ABB RobotStudio station: Minor Project_Kundan_Singh_48849855.rspag

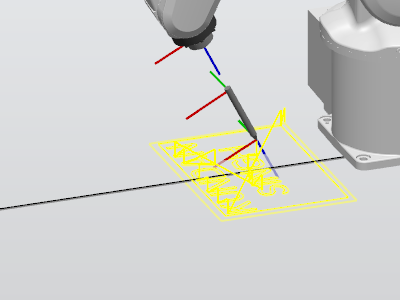
--- station ---
Station Minor Project Kundan1_4 (saved by RobotStudio 23.2.10395.0)
Controller Controller8, task T_ROB1: task frame (RAPID world) sits at (0, -187, 16) mm in the station
Controller Controller8
  mechanical unit ROB_1: IRB120_3_58__01, 6 joints, base frame (0, 0, 0) mm
Layout (positions relative to the parent item):
  - IRB120_3_58__01 [mechanism, from %ABB.RobotStudio.Models.IRB120%\IRB120_3_58_G_01.rslib] at (0, -187, 16) mm; joint values [-1.7305, 0.6039, 0.6241, -0.0997, 0.8114, 3.0678] (rad or m)
  - CaliCone [part], size 200 x 198.5 x 250 mm
  - Table [part], size 250 x 500 x 250 mm
  - A4 [part], size 210 x 297 x 0.4 mm
  - a4_border_name [part] at (404.58, 0, 250) mm, rotated rx 90 ry 0 rz -90 deg, size 277 x 2 x 190 mm
  - My_Mechanism [mechanism] at (-51.03, -471, 203.2) mm, rotated rx -180 ry 27 rz -90 deg; joint values [-0.1] (rad or m)
      TCP My_Mechanism_1 at (0, 163.83, 0) mm, rotated rx -90 ry 0 rz 0 deg
      links: base, L1
  - Frame_1 [frame] at (0, 0, 100) mm
Attachment: My_Mechanism is attached to IRB120_3_58__01 / Link6
Targets, tools, work objects and paths stored in the station and not in the controller backup, written as RAPID:
! task T_ROB1
MODULE Module1
  CONST robtarget Target_20_2:=[[323,-148.5,7.4],[0,0.97236992,0,-0.233445365],[-2,-1,1,0],[9E+09,9E+09,9E+09,9E+09,9E+09,9E+09]];
  CONST robtarget Target_30_2:=[[323,148.5,7.4],[0,0.97236992,0,-0.233445365],[-1,0,2,0],[9E+09,9E+09,9E+09,9E+09,9E+09,9E+09]];
  CONST robtarget Target_40_2:=[[113,148.5,7.4],[0,0.97236992,0,-0.233445365],[-1,0,2,0],[9E+09,9E+09,9E+09,9E+09,9E+09,9E+09]];
ENDMODULE


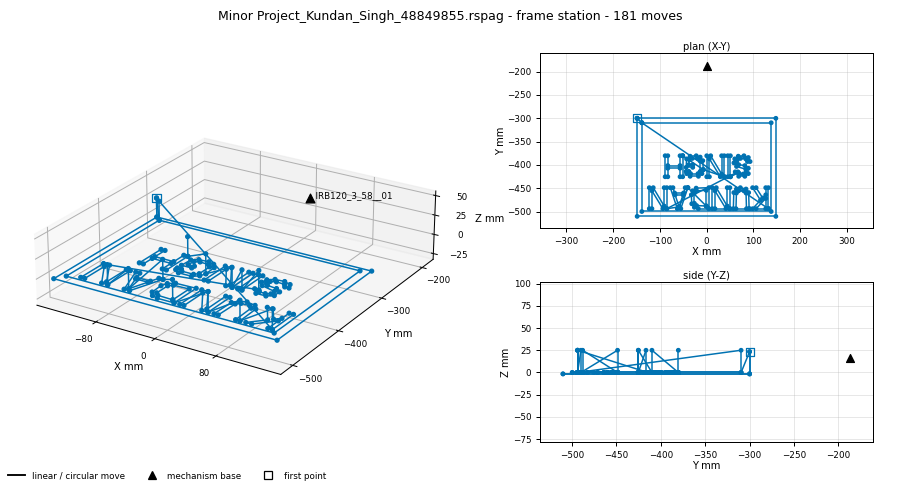
[picture p0: tool path of Minor Project_Kundan_Singh_48849855.rspag in frame station, 181 of 181 moves have a stored position in this frame; points joined in program order, loops and branches not executed]
--- Backups/Controller8/RAPID/TASK1/PROGMOD/CalibData.mod ---
MODULE CalibData
    TASK PERS wobjdata Minor_1:=[FALSE,TRUE,"",[[0,0,0],[0.707106781,0,0,-0.707106781]],[[0,0,0],[1,0,0,0]]];
ENDMODULE

--- Backups/Controller8/RAPID/TASK1/PROGMOD/Module1.mod ---
MODULE Module1
    TASK PERS tooldata TCP_Manual:=[TRUE,[[-0.00301652,0.0402778,105.238],[0.999972622,-0.000427662,-0.004756351,-0.005652456]],[1,[1,0,0],[1,0,0,0],0,0,0]];
    PERS tooldata My_Mechanism_2:=[TRUE,[[0,0,200],[1,0,0,0]],[1,[1,0,0],[1,0,0,0],0,0,0]];
    CONST robtarget Target_10_2:=[[113,-148.5,7.4],[0,0.97236992,0,-0.233445365],[-2,-1,1,0],[9E+09,9E+09,9E+09,9E+09,9E+09,9E+09]];
    CONST robtarget Target_10:=[[113,-148.5,-17.6],[0,0.97236992,0,-0.233445365],[-2,-1,1,0],[9E+09,9E+09,9E+09,9E+09,9E+09,9E+09]];
    CONST robtarget Target_20:=[[323,-148.5,-17.6],[0,0.97236992,0,-0.233445365],[-2,-1,1,0],[9E+09,9E+09,9E+09,9E+09,9E+09,9E+09]];
    CONST robtarget Target_30:=[[323,148.5,-17.6],[0,0.97236992,0,-0.233445365],[-1,0,2,0],[9E+09,9E+09,9E+09,9E+09,9E+09,9E+09]];
    CONST robtarget Target_40:=[[113,148.5,-17.6],[0,0.97236992,0,-0.233445365],[-1,0,2,0],[9E+09,9E+09,9E+09,9E+09,9E+09,9E+09]];
    CONST robtarget Target_50:=[[113,-148.5,-17.6],[0,0.97236992,0,-0.233445365],[-2,-1,1,0],[9E+09,9E+09,9E+09,9E+09,9E+09,9E+09]];
    CONST robtarget Target_60:=[[122.583914519,-138.5,-16],[0,0.97236992,0,-0.233445365],[-2,-1,1,0],[9E+09,9E+09,9E+09,9E+09,9E+09,9E+09]];
    CONST robtarget Target_70:=[[312.583914519,-138.5,-16],[0,0.97236992,0,-0.233445365],[-2,-1,1,0],[9E+09,9E+09,9E+09,9E+09,9E+09,9E+09]];
    CONST robtarget Target_80:=[[312.583914519,138.5,-16],[0,0.97236992,0,-0.233445365],[-1,0,2,0],[9E+09,9E+09,9E+09,9E+09,9E+09,9E+09]];
    CONST robtarget Target_90:=[[122.583914519,138.5,-16],[0,0.97236992,0,-0.233445365],[-1,0,2,0],[9E+09,9E+09,9E+09,9E+09,9E+09,9E+09]];
    CONST robtarget Target_100:=[[122.583914519,-138.5,-16],[0,0.97236992,0,-0.233445365],[-2,-1,1,0],[9E+09,9E+09,9E+09,9E+09,9E+09,9E+09]];
    CONST robtarget Target_100_2:=[[122.583914519,-138.5,9],[0,0.97236992,0,-0.233445365],[-2,-1,1,0],[9E+09,9E+09,9E+09,9E+09,9E+09,9E+09]];
    CONST robtarget Target_110:=[[306.583914519,132.5,-16],[0,0.97236992,0,-0.233445365],[-1,0,2,0],[9E+09,9E+09,9E+09,9E+09,9E+09,9E+09]];
    CONST robtarget Target_120:=[[261.583914519,132.5,-16],[0,0.97236992,0,-0.233445365],[-1,0,2,0],[9E+09,9E+09,9E+09,9E+09,9E+09,9E+09]];
    CONST robtarget Target_130:=[[261.583914519,126.875,-16],[0,0.97236992,0,-0.233445365],[-1,0,2,0],[9E+09,9E+09,9E+09,9E+09,9E+09,9E+09]];
    CONST robtarget Target_140:=[[276.903062971,126.875,-16],[0,0.97236992,0,-0.233445365],[-1,0,2,0],[9E+09,9E+09,9E+09,9E+09,9E+09,9E+09]];
    CONST robtarget Target_150:=[[283.605191172,120.312499553,-16],[0,0.97236992,0,-0.233445365],[-1,0,2,0],[9E+09,9E+09,9E+09,9E+09,9E+09,9E+09]];
    CONST robtarget Target_160:=[[261.583914519,106.250000894,-16],[0,0.97236992,0,-0.233445365],[-1,0,2,0],[9E+09,9E+09,9E+09,9E+09,9E+09,9E+09]];
    CONST robtarget Target_170:=[[261.583914519,98.75,-16],[0,0.97236992,0,-0.233445365],[-1,0,2,0],[9E+09,9E+09,9E+09,9E+09,9E+09,9E+09]];
    CONST robtarget Target_180:=[[288.392424644,115.625,-16],[0,0.97236992,0,-0.233445365],[-1,0,2,0],[9E+09,9E+09,9E+09,9E+09,9E+09,9E+09]];
    CONST robtarget Target_190:=[[306.583914519,98.75,-16],[0,0.97236992,0,-0.233445365],[-1,0,2,0],[9E+09,9E+09,9E+09,9E+09,9E+09,9E+09]];
    CONST robtarget Target_200:=[[306.583914519,106.250000894,-16],[0,0.97236992,0,-0.233445365],[-1,0,2,0],[9E+09,9E+09,9E+09,9E+09,9E+09,9E+09]];
    CONST robtarget Target_210:=[[284.562637867,126.875,-16],[0,0.97236992,0,-0.233445365],[-1,0,2,0],[9E+09,9E+09,9E+09,9E+09,9E+09,9E+09]];
    CONST robtarget Target_220:=[[306.583914519,126.875,-16],[0,0.97236992,0,-0.233445365],[-1,0,2,0],[9E+09,9E+09,9E+09,9E+09,9E+09,9E+09]];
    CONST robtarget Target_230:=[[306.583914519,132.5,-16],[0,0.97236992,0,-0.233445365],[-1,0,2,0],[9E+09,9E+09,9E+09,9E+09,9E+09,9E+09]];
    CONST robtarget Target_230_2:=[[306.583914519,132.5,9],[0,0.97236992,0,-0.233445365],[-1,0,2,0],[9E+09,9E+09,9E+09,9E+09,9E+09,9E+09]];
    CONST robtarget Target_240:=[[306.583914519,91.249999106,-16],[0,0.97236992,0,-0.233445365],[-1,0,2,0],[9E+09,9E+09,9E+09,9E+09,9E+09,9E+09]];
    CONST robtarget Target_250:=[[272.115829499,90.3125,-16],[0,0.97236992,0,-0.233445365],[-1,0,2,0],[9E+09,9E+09,9E+09,9E+09,9E+09,9E+09]];
    CONST robtarget Target_260:=[[264.456254938,84.6875,-16],[0,0.97236992,0,-0.233445365],[-1,0,2,0],[9E+09,9E+09,9E+09,9E+09,9E+09,9E+09]];
    CONST robtarget Target_270:=[[261.583914519,72.499998212,-16],[0,0.97236992,0,-0.233445365],[-1,0,2,0],[9E+09,9E+09,9E+09,9E+09,9E+09,9E+09]];
    CONST robtarget Target_280:=[[264.456254938,64.062498212,-16],[0,0.97236992,0,-0.233445365],[-1,0,2,0],[9E+09,9E+09,9E+09,9E+09,9E+09,9E+09]];
    CONST robtarget Target_290:=[[272.115829499,58.437498212,-16],[0,0.97236992,0,-0.233445365],[-1,0,2,0],[9E+09,9E+09,9E+09,9E+09,9E+09,9E+09]];
    CONST robtarget Target_300:=[[306.583914519,57.500001788,-16],[0,0.97236992,0,-0.233445365],[-1,0,2,0],[9E+09,9E+09,9E+09,9E+09,9E+09,9E+09]];
    CONST robtarget Target_310:=[[306.583914519,63.125001788,-16],[0,0.97236992,0,-0.233445365],[-1,0,2,0],[9E+09,9E+09,9E+09,9E+09,9E+09,9E+09]];
    CONST robtarget Target_320:=[[273.073276193,64.062498212,-16],[0,0.97236992,0,-0.233445365],[-1,0,2,0],[9E+09,9E+09,9E+09,9E+09,9E+09,9E+09]];
    CONST robtarget Target_330:=[[268.286042051,68.750001788,-16],[0,0.97236992,0,-0.233445365],[-1,0,2,0],[9E+09,9E+09,9E+09,9E+09,9E+09,9E+09]];
    CONST robtarget Target_340:=[[268.286042051,80.000001788,-16],[0,0.97236992,0,-0.233445365],[-1,0,2,0],[9E+09,9E+09,9E+09,9E+09,9E+09,9E+09]];
    CONST robtarget Target_350:=[[273.073276193,84.6875,-16],[0,0.97236992,0,-0.233445365],[-1,0,2,0],[9E+09,9E+09,9E+09,9E+09,9E+09,9E+09]];
    CONST robtarget Target_360:=[[306.583914519,85.625001788,-16],[0,0.97236992,0,-0.233445365],[-1,0,2,0],[9E+09,9E+09,9E+09,9E+09,9E+09,9E+09]];
    CONST robtarget Target_370:=[[306.583914519,91.249999106,-16],[0,0.97236992,0,-0.233445365],[-1,0,2,0],[9E+09,9E+09,9E+09,9E+09,9E+09,9E+09]];
    CONST robtarget Target_370_2:=[[306.583914519,91.249999106,9],[0,0.97236992,0,-0.233445365],[-1,0,2,0],[9E+09,9E+09,9E+09,9E+09,9E+09,9E+09]];
    CONST robtarget Target_380:=[[306.583914519,49.999998212,-16],[0,0.97236992,0,-0.233445365],[-1,0,2,0],[9E+09,9E+09,9E+09,9E+09,9E+09,9E+09]];
    CONST robtarget Target_390:=[[261.583914519,49.999998212,-16],[0,0.97236992,0,-0.233445365],[-1,0,2,0],[9E+09,9E+09,9E+09,9E+09,9E+09,9E+09]];
    CONST robtarget Target_400:=[[261.583914519,44.374998212,-16],[0,0.97236992,0,-0.233445365],[-1,0,2,0],[9E+09,9E+09,9E+09,9E+09,9E+09,9E+09]];
    CONST robtarget Target_410:=[[300.839234353,44.374998212,-16],[0,0.97236992,0,-0.233445365],[-1,0,2,0],[9E+09,9E+09,9E+09,9E+09,9E+09,9E+09]];
    CONST robtarget Target_420:=[[261.583914519,20.937496424,-16],[0,0.97236992,0,-0.233445365],[-1,0,2,0],[9E+09,9E+09,9E+09,9E+09,9E+09,9E+09]];
    CONST robtarget Target_430:=[[261.583914519,12.499996424,-16],[0,0.97236992,0,-0.233445365],[-1,0,2,0],[9E+09,9E+09,9E+09,9E+09,9E+09,9E+09]];
    CONST robtarget Target_440:=[[306.583914519,12.499996424,-16],[0,0.97236992,0,-0.233445365],[-1,0,2,0],[9E+09,9E+09,9E+09,9E+09,9E+09,9E+09]];
    CONST robtarget Target_450:=[[306.583914519,18.124996424,-16],[0,0.97236992,0,-0.233445365],[-1,0,2,0],[9E+09,9E+09,9E+09,9E+09,9E+09,9E+09]];
    CONST robtarget Target_460:=[[268.286042051,18.124996424,-16],[0,0.97236992,0,-0.233445365],[-1,0,2,0],[9E+09,9E+09,9E+09,9E+09,9E+09,9E+09]];
    CONST robtarget Target_470:=[[306.583914519,41.562503576,-16],[0,0.97236992,0,-0.233445365],[-1,0,2,0],[9E+09,9E+09,9E+09,9E+09,9E+09,9E+09]];
    CONST robtarget Target_480:=[[306.583914519,49.999998212,-16],[0,0.97236992,0,-0.233445365],[-1,0,2,0],[9E+09,9E+09,9E+09,9E+09,9E+09,9E+09]];
    CONST robtarget Target_480_2:=[[306.583914519,49.999998212,9],[0,0.97236992,0,-0.233445365],[-1,0,2,0],[9E+09,9E+09,9E+09,9E+09,9E+09,9E+09]];
    CONST robtarget Target_490:=[[306.583914519,5.000003576,-16],[0,0.97236992,0,-0.233445365],[-1,0,2,0],[9E+09,9E+09,9E+09,9E+09,9E+09,9E+09]];
    CONST robtarget Target_500:=[[261.583914519,5.000003576,-16],[0,0.97236992,0,-0.233445365],[-1,0,2,0],[9E+09,9E+09,9E+09,9E+09,9E+09,9E+09]];
    CONST robtarget Target_510:=[[262.541361298,-22.1875,-16],[0,0.97236992,0,-0.233445365],[-2,-1,1,0],[9E+09,9E+09,9E+09,9E+09,9E+09,9E+09]];
    CONST robtarget Target_520:=[[268.286042051,-29.687503576,-16],[0,0.97236992,0,-0.233445365],[-2,-1,1,0],[9E+09,9E+09,9E+09,9E+09,9E+09,9E+09]];
    CONST robtarget Target_530:=[[276.903062971,-32.500003576,-16],[0,0.97236992,0,-0.233445365],[-2,-1,1,0],[9E+09,9E+09,9E+09,9E+09,9E+09,9E+09]];
    CONST robtarget Target_540:=[[296.052000881,-31.562496424,-16],[0,0.97236992,0,-0.233445365],[-2,-1,1,0],[9E+09,9E+09,9E+09,9E+09,9E+09,9E+09]];
    CONST robtarget Target_550:=[[303.711574436,-25.937496424,-16],[0,0.97236992,0,-0.233445365],[-2,-1,1,0],[9E+09,9E+09,9E+09,9E+09,9E+09,9E+09]];
    CONST robtarget Target_560:=[[306.583914519,-17.499996424,-16],[0,0.97236992,0,-0.233445365],[-2,-1,1,0],[9E+09,9E+09,9E+09,9E+09,9E+09,9E+09]];
    CONST robtarget Target_570:=[[306.583914519,5.000003576,-16],[0,0.97236992,0,-0.233445365],[-1,0,2,0],[9E+09,9E+09,9E+09,9E+09,9E+09,9E+09]];
    CONST robtarget Target_580:=[[300.839234353,-0.624996424,-16],[0,0.97236992,0,-0.233445365],[-2,-1,1,0],[9E+09,9E+09,9E+09,9E+09,9E+09,9E+09]];
    CONST robtarget Target_580_2:=[[300.839234353,-0.624996424,9],[0,0.97236992,0,-0.233445365],[-2,-1,1,0],[9E+09,9E+09,9E+09,9E+09,9E+09,9E+09]];
    CONST robtarget Target_590:=[[267.328595356,-0.624996424,-16],[0,0.97236992,0,-0.233445365],[-2,-1,1,0],[9E+09,9E+09,9E+09,9E+09,9E+09,9E+09]];
    CONST robtarget Target_600:=[[268.286042051,-21.250003576,-16],[0,0.97236992,0,-0.233445365],[-2,-1,1,0],[9E+09,9E+09,9E+09,9E+09,9E+09,9E+09]];
    CONST robtarget Target_610:=[[273.073276193,-25.937496424,-16],[0,0.97236992,0,-0.233445365],[-2,-1,1,0],[9E+09,9E+09,9E+09,9E+09,9E+09,9E+09]];
    CONST robtarget Target_620:=[[295.094551505,-25.937496424,-16],[0,0.97236992,0,-0.233445365],[-2,-1,1,0],[9E+09,9E+09,9E+09,9E+09,9E+09,9E+09]];
    CONST robtarget Target_630:=[[299.881787659,-21.250003576,-16],[0,0.97236992,0,-0.233445365],[-2,-1,1,0],[9E+09,9E+09,9E+09,9E+09,9E+09,9E+09]];
    CONST robtarget Target_640:=[[300.839234353,-0.624996424,-16],[0,0.97236992,0,-0.233445365],[-2,-1,1,0],[9E+09,9E+09,9E+09,9E+09,9E+09,9E+09]];
    CONST robtarget Target_640_2:=[[300.839234353,-0.624996424,9],[0,0.97236992,0,-0.233445365],[-2,-1,1,0],[9E+09,9E+09,9E+09,9E+09,9E+09,9E+09]];
    CONST robtarget Target_650:=[[261.583914519,-39.999996424,-16],[0,0.97236992,0,-0.233445365],[-2,-1,1,0],[9E+09,9E+09,9E+09,9E+09,9E+09,9E+09]];
    CONST robtarget Target_660:=[[306.583914519,-54.999992847,-16],[0,0.97236992,0,-0.233445365],[-2,-1,1,0],[9E+09,9E+09,9E+09,9E+09,9E+09,9E+09]];
    CONST robtarget Target_670:=[[306.583914519,-62.500007153,-16],[0,0.97236992,0,-0.233445365],[-2,-1,1,0],[9E+09,9E+09,9E+09,9E+09,9E+09,9E+09]];
    CONST robtarget Target_680:=[[261.583914519,-77.499992847,-16],[0,0.97236992,0,-0.233445365],[-2,-1,1,0],[9E+09,9E+09,9E+09,9E+09,9E+09,9E+09]];
    CONST robtarget Target_690:=[[261.583914519,-71.874992847,-16],[0,0.97236992,0,-0.233445365],[-2,-1,1,0],[9E+09,9E+09,9E+09,9E+09,9E+09,9E+09]];
    CONST robtarget Target_700:=[[273.073276193,-68.125007153,-16],[0,0.97236992,0,-0.233445365],[-2,-1,1,0],[9E+09,9E+09,9E+09,9E+09,9E+09,9E+09]];
    CONST robtarget Target_710:=[[273.073276193,-49.374992847,-16],[0,0.97236992,0,-0.233445365],[-2,-1,1,0],[9E+09,9E+09,9E+09,9E+09,9E+09,9E+09]];
    CONST robtarget Target_720:=[[261.583914519,-45.624996424,-16],[0,0.97236992,0,-0.233445365],[-2,-1,1,0],[9E+09,9E+09,9E+09,9E+09,9E+09,9E+09]];
    CONST robtarget Target_730:=[[261.583914519,-39.999996424,-16],[0,0.97236992,0,-0.233445365],[-2,-1,1,0],[9E+09,9E+09,9E+09,9E+09,9E+09,9E+09]];
    CONST robtarget Target_730_2:=[[261.583914519,-39.999996424,9],[0,0.97236992,0,-0.233445365],[-2,-1,1,0],[9E+09,9E+09,9E+09,9E+09,9E+09,9E+09]];
    CONST robtarget Target_740:=[[302.754127742,-58.75,-16],[0,0.97236992,0,-0.233445365],[-2,-1,1,0],[9E+09,9E+09,9E+09,9E+09,9E+09,9E+09]];
    CONST robtarget Target_750:=[[276.903062971,-50.3125,-16],[0,0.97236992,0,-0.233445365],[-2,-1,1,0],[9E+09,9E+09,9E+09,9E+09,9E+09,9E+09]];
    CONST robtarget Target_760:=[[276.903062971,-67.1875,-16],[0,0.97236992,0,-0.233445365],[-2,-1,1,0],[9E+09,9E+09,9E+09,9E+09,9E+09,9E+09]];
    CONST robtarget Target_770:=[[302.754127742,-58.75,-16],[0,0.97236992,0,-0.233445365],[-2,-1,1,0],[9E+09,9E+09,9E+09,9E+09,9E+09,9E+09]];
    CONST robtarget Target_770_2:=[[302.754127742,-58.75,9],[0,0.97236992,0,-0.233445365],[-2,-1,1,0],[9E+09,9E+09,9E+09,9E+09,9E+09,9E+09]];
    CONST robtarget Target_780:=[[306.583914519,-85.000007153,-16],[0,0.97236992,0,-0.233445365],[-2,-1,1,0],[9E+09,9E+09,9E+09,9E+09,9E+09,9E+09]];
    CONST robtarget Target_790:=[[261.583914519,-85.000007153,-16],[0,0.97236992,0,-0.233445365],[-2,-1,1,0],[9E+09,9E+09,9E+09,9E+09,9E+09,9E+09]];
    CONST robtarget Target_800:=[[261.583914519,-90.625007153,-16],[0,0.97236992,0,-0.233445365],[-2,-1,1,0],[9E+09,9E+09,9E+09,9E+09,9E+09,9E+09]];
    CONST robtarget Target_810:=[[300.839234353,-90.625007153,-16],[0,0.97236992,0,-0.233445365],[-2,-1,1,0],[9E+09,9E+09,9E+09,9E+09,9E+09,9E+09]];
    CONST robtarget Target_820:=[[261.583914519,-114.062492847,-16],[0,0.97236992,0,-0.233445365],[-2,-1,1,0],[9E+09,9E+09,9E+09,9E+09,9E+09,9E+09]];
    CONST robtarget Target_830:=[[261.583914519,-122.499992847,-16],[0,0.97236992,0,-0.233445365],[-2,-1,1,0],[9E+09,9E+09,9E+09,9E+09,9E+09,9E+09]];
    CONST robtarget Target_840:=[[306.583914519,-122.499992847,-16],[0,0.97236992,0,-0.233445365],[-2,-1,1,0],[9E+09,9E+09,9E+09,9E+09,9E+09,9E+09]];
    CONST robtarget Target_850:=[[306.583914519,-116.874992847,-16],[0,0.97236992,0,-0.233445365],[-2,-1,1,0],[9E+09,9E+09,9E+09,9E+09,9E+09,9E+09]];
    CONST robtarget Target_860:=[[268.286042051,-116.874992847,-16],[0,0.97236992,0,-0.233445365],[-2,-1,1,0],[9E+09,9E+09,9E+09,9E+09,9E+09,9E+09]];
    CONST robtarget Target_870:=[[306.583914519,-93.437507153,-16],[0,0.97236992,0,-0.233445365],[-2,-1,1,0],[9E+09,9E+09,9E+09,9E+09,9E+09,9E+09]];
    CONST robtarget Target_880:=[[306.583914519,-85.000007153,-16],[0,0.97236992,0,-0.233445365],[-2,-1,1,0],[9E+09,9E+09,9E+09,9E+09,9E+09,9E+09]];
    CONST robtarget Target_880_2:=[[306.583914519,-85.000007153,9],[0,0.97236992,0,-0.233445365],[-2,-1,1,0],[9E+09,9E+09,9E+09,9E+09,9E+09,9E+09]];
    CONST robtarget Target_890:=[[227.667879541,67.099183578,-16],[0,0.97236992,0,-0.233445365],[-1,0,2,0],[9E+09,9E+09,9E+09,9E+09,9E+09,9E+09]];
    CONST robtarget Target_900:=[[227.667879541,61.474183578,-16],[0,0.97236992,0,-0.233445365],[-1,0,2,0],[9E+09,9E+09,9E+09,9E+09,9E+09,9E+09]];
    CONST robtarget Target_910:=[[237.242346485,68.974181789,-16],[0,0.97236992,0,-0.233445365],[-1,0,2,0],[9E+09,9E+09,9E+09,9E+09,9E+09,9E+09]];
    CONST robtarget Target_920:=[[237.242346485,82.099182684,-16],[0,0.97236992,0,-0.233445365],[-1,0,2,0],[9E+09,9E+09,9E+09,9E+09,9E+09,9E+09]];
    CONST robtarget Target_930:=[[231.497666319,89.599182572,-16],[0,0.97236992,0,-0.233445365],[-1,0,2,0],[9E+09,9E+09,9E+09,9E+09,9E+09,9E+09]];
    CONST robtarget Target_940:=[[220.008303304,89.599182572,-16],[0,0.97236992,0,-0.233445365],[-1,0,2,0],[9E+09,9E+09,9E+09,9E+09,9E+09,9E+09]];
    CONST robtarget Target_950:=[[214.263623138,82.099182684,-16],[0,0.97236992,0,-0.233445365],[-1,0,2,0],[9E+09,9E+09,9E+09,9E+09,9E+09,9E+09]];
    CONST robtarget Target_960:=[[212.348729749,68.974181789,-16],[0,0.97236992,0,-0.233445365],[-1,0,2,0],[9E+09,9E+09,9E+09,9E+09,9E+09,9E+09]];
    CONST robtarget Target_970:=[[207.561494936,64.286683578,-16],[0,0.97236992,0,-0.233445365],[-1,0,2,0],[9E+09,9E+09,9E+09,9E+09,9E+09,9E+09]];
    CONST robtarget Target_980:=[[201.81681477,66.161681789,-16],[0,0.97236992,0,-0.233445365],[-1,0,2,0],[9E+09,9E+09,9E+09,9E+09,9E+09,9E+09]];
    CONST robtarget Target_990:=[[198.944474016,72.724182236,-16],[0,0.97236992,0,-0.233445365],[-1,0,2,0],[9E+09,9E+09,9E+09,9E+09,9E+09,9E+09]];
    CONST robtarget Target_1000:=[[199.901920711,83.974182907,-16],[0,0.97236992,0,-0.233445365],[-1,0,2,0],[9E+09,9E+09,9E+09,9E+09,9E+09,9E+09]];
    CONST robtarget Target_1010:=[[205.646601547,87.724182684,-16],[0,0.97236992,0,-0.233445365],[-1,0,2,0],[9E+09,9E+09,9E+09,9E+09,9E+09,9E+09]];
    CONST robtarget Target_1020:=[[205.646601547,93.349182684,-16],[0,0.97236992,0,-0.233445365],[-1,0,2,0],[9E+09,9E+09,9E+09,9E+09,9E+09,9E+09]];
    CONST robtarget Target_1030:=[[197.029580292,89.599182572,-16],[0,0.97236992,0,-0.233445365],[-1,0,2,0],[9E+09,9E+09,9E+09,9E+09,9E+09,9E+09]];
    CONST robtarget Target_1040:=[[193.199793179,80.224183131,-16],[0,0.97236992,0,-0.233445365],[-1,0,2,0],[9E+09,9E+09,9E+09,9E+09,9E+09,9E+09]];
    CONST robtarget Target_1050:=[[194.157239958,68.036682684,-16],[0,0.97236992,0,-0.233445365],[-1,0,2,0],[9E+09,9E+09,9E+09,9E+09,9E+09,9E+09]];
    CONST robtarget Target_1060:=[[199.901920711,60.536681789,-16],[0,0.97236992,0,-0.233445365],[-1,0,2,0],[9E+09,9E+09,9E+09,9E+09,9E+09,9E+09]];
    CONST robtarget Target_1070:=[[208.51894163,58.661683578,-16],[0,0.97236992,0,-0.233445365],[-1,0,2,0],[9E+09,9E+09,9E+09,9E+09,9E+09,9E+09]];
    CONST robtarget Target_1080:=[[216.178516527,64.286683578,-16],[0,0.97236992,0,-0.233445365],[-1,0,2,0],[9E+09,9E+09,9E+09,9E+09,9E+09,9E+09]];
    CONST robtarget Target_1090:=[[221.923196693,83.974182907,-16],[0,0.97236992,0,-0.233445365],[-1,0,2,0],[9E+09,9E+09,9E+09,9E+09,9E+09,9E+09]];
    CONST robtarget Target_1100:=[[229.58277293,83.974182907,-16],[0,0.97236992,0,-0.233445365],[-1,0,2,0],[9E+09,9E+09,9E+09,9E+09,9E+09,9E+09]];
    CONST robtarget Target_1110:=[[232.455113013,78.349182236,-16],[0,0.97236992,0,-0.233445365],[-1,0,2,0],[9E+09,9E+09,9E+09,9E+09,9E+09,9E+09]];
    CONST robtarget Target_1120:=[[231.497666319,69.911683578,-16],[0,0.97236992,0,-0.233445365],[-1,0,2,0],[9E+09,9E+09,9E+09,9E+09,9E+09,9E+09]];
    CONST robtarget Target_1130:=[[229.58277293,68.036682684,-16],[0,0.97236992,0,-0.233445365],[-1,0,2,0],[9E+09,9E+09,9E+09,9E+09,9E+09,9E+09]];
    CONST robtarget Target_1130_2:=[[229.58277293,68.036682684,9],[0,0.97236992,0,-0.233445365],[-1,0,2,0],[9E+09,9E+09,9E+09,9E+09,9E+09,9E+09]];
    CONST robtarget Target_1140:=[[238.199793179,51.161682684,-16],[0,0.97236992,0,-0.233445365],[-1,0,2,0],[9E+09,9E+09,9E+09,9E+09,9E+09,9E+09]];
    CONST robtarget Target_1150:=[[193.199793179,51.161682684,-16],[0,0.97236992,0,-0.233445365],[-1,0,2,0],[9E+09,9E+09,9E+09,9E+09,9E+09,9E+09]];
    CONST robtarget Target_1160:=[[193.199793179,45.536682684,-16],[0,0.97236992,0,-0.233445365],[-1,0,2,0],[9E+09,9E+09,9E+09,9E+09,9E+09,9E+09]];
    CONST robtarget Target_1170:=[[238.199793179,45.536682684,-16],[0,0.97236992,0,-0.233445365],[-1,0,2,0],[9E+09,9E+09,9E+09,9E+09,9E+09,9E+09]];
    CONST robtarget Target_1180:=[[238.199793179,51.161682684,-16],[0,0.97236992,0,-0.233445365],[-1,0,2,0],[9E+09,9E+09,9E+09,9E+09,9E+09,9E+09]];
    CONST robtarget Target_1180_2:=[[238.199793179,51.161682684,9],[0,0.97236992,0,-0.233445365],[-1,0,2,0],[9E+09,9E+09,9E+09,9E+09,9E+09,9E+09]];
    CONST robtarget Target_1190:=[[238.199793179,38.036684472,-16],[0,0.97236992,0,-0.233445365],[-1,0,2,0],[9E+09,9E+09,9E+09,9E+09,9E+09,9E+09]];
    CONST robtarget Target_1200:=[[193.199793179,38.036684472,-16],[0,0.97236992,0,-0.233445365],[-1,0,2,0],[9E+09,9E+09,9E+09,9E+09,9E+09,9E+09]];
    CONST robtarget Target_1210:=[[193.199793179,32.411684472,-16],[0,0.97236992,0,-0.233445365],[-1,0,2,0],[9E+09,9E+09,9E+09,9E+09,9E+09,9E+09]];
    CONST robtarget Target_1220:=[[232.455113013,32.411684472,-16],[0,0.97236992,0,-0.233445365],[-1,0,2,0],[9E+09,9E+09,9E+09,9E+09,9E+09,9E+09]];
    CONST robtarget Target_1230:=[[193.199793179,8.974182684,-16],[0,0.97236992,0,-0.233445365],[-1,0,2,0],[9E+09,9E+09,9E+09,9E+09,9E+09,9E+09]];
    CONST robtarget Target_1240:=[[193.199793179,0.536682684,-16],[0,0.97236992,0,-0.233445365],[-1,0,2,0],[9E+09,9E+09,9E+09,9E+09,9E+09,9E+09]];
    CONST robtarget Target_1250:=[[238.199793179,0.536682684,-16],[0,0.97236992,0,-0.233445365],[-1,0,2,0],[9E+09,9E+09,9E+09,9E+09,9E+09,9E+09]];
    CONST robtarget Target_1260:=[[238.199793179,6.161682684,-16],[0,0.97236992,0,-0.233445365],[-1,0,2,0],[9E+09,9E+09,9E+09,9E+09,9E+09,9E+09]];
    CONST robtarget Target_1270:=[[199.901920711,6.161682684,-16],[0,0.97236992,0,-0.233445365],[-1,0,2,0],[9E+09,9E+09,9E+09,9E+09,9E+09,9E+09]];
    CONST robtarget Target_1280:=[[238.199793179,29.599184472,-16],[0,0.97236992,0,-0.233445365],[-1,0,2,0],[9E+09,9E+09,9E+09,9E+09,9E+09,9E+09]];
    CONST robtarget Target_1290:=[[238.199793179,38.036684472,-16],[0,0.97236992,0,-0.233445365],[-1,0,2,0],[9E+09,9E+09,9E+09,9E+09,9E+09,9E+09]];
    CONST robtarget Target_1290_2:=[[238.199793179,38.036684472,9],[0,0.97236992,0,-0.233445365],[-1,0,2,0],[9E+09,9E+09,9E+09,9E+09,9E+09,9E+09]];
    CONST robtarget Target_1300:=[[222.880643387,-6.963320893,-16],[0,0.97236992,0,-0.233445365],[-2,-1,1,0],[9E+09,9E+09,9E+09,9E+09,9E+09,9E+09]];
    CONST robtarget Target_1310:=[[203.731708159,-7.900817316,-16],[0,0.97236992,0,-0.233445365],[-2,-1,1,0],[9E+09,9E+09,9E+09,9E+09,9E+09,9E+09]];
    CONST robtarget Target_1320:=[[196.072133598,-13.525817316,-16],[0,0.97236992,0,-0.233445365],[-2,-1,1,0],[9E+09,9E+09,9E+09,9E+09,9E+09,9E+09]];
    CONST robtarget Target_1330:=[[193.199793179,-21.963317316,-16],[0,0.97236992,0,-0.233445365],[-2,-1,1,0],[9E+09,9E+09,9E+09,9E+09,9E+09,9E+09]];
    CONST robtarget Target_1340:=[[194.157239958,-35.088320893,-16],[0,0.97236992,0,-0.233445365],[-2,-1,1,0],[9E+09,9E+09,9E+09,9E+09,9E+09,9E+09]];
    CONST robtarget Target_1350:=[[199.901920711,-42.58831374,-16],[0,0.97236992,0,-0.233445365],[-2,-1,1,0],[9E+09,9E+09,9E+09,9E+09,9E+09,9E+09]];
    CONST robtarget Target_1360:=[[218.093409915,-43.525820893,-16],[0,0.97236992,0,-0.233445365],[-2,-1,1,0],[9E+09,9E+09,9E+09,9E+09,9E+09,9E+09]];
    CONST robtarget Target_1370:=[[218.093409915,-29.463320893,-16],[0,0.97236992,0,-0.233445365],[-2,-1,1,0],[9E+09,9E+09,9E+09,9E+09,9E+09,9E+09]];
    CONST robtarget Target_1380:=[[212.348729749,-29.463320893,-16],[0,0.97236992,0,-0.233445365],[-2,-1,1,0],[9E+09,9E+09,9E+09,9E+09,9E+09,9E+09]];
    CONST robtarget Target_1390:=[[212.348729749,-37.900820893,-16],[0,0.97236992,0,-0.233445365],[-2,-1,1,0],[9E+09,9E+09,9E+09,9E+09,9E+09,9E+09]];
    CONST robtarget Target_1400:=[[201.81681477,-36.96331374,-16],[0,0.97236992,0,-0.233445365],[-2,-1,1,0],[9E+09,9E+09,9E+09,9E+09,9E+09,9E+09]];
    CONST robtarget Target_1410:=[[198.944474016,-30.400817316,-16],[0,0.97236992,0,-0.233445365],[-2,-1,1,0],[9E+09,9E+09,9E+09,9E+09,9E+09,9E+09]];
    CONST robtarget Target_1420:=[[199.901920711,-18.213320893,-16],[0,0.97236992,0,-0.233445365],[-2,-1,1,0],[9E+09,9E+09,9E+09,9E+09,9E+09,9E+09]];
    CONST robtarget Target_1430:=[[204.689154853,-13.525817316,-16],[0,0.97236992,0,-0.233445365],[-2,-1,1,0],[9E+09,9E+09,9E+09,9E+09,9E+09,9E+09]];
    CONST robtarget Target_1440:=[[226.710430165,-13.525817316,-16],[0,0.97236992,0,-0.233445365],[-2,-1,1,0],[9E+09,9E+09,9E+09,9E+09,9E+09,9E+09]];
    CONST robtarget Target_1450:=[[231.497666319,-18.213320893,-16],[0,0.97236992,0,-0.233445365],[-2,-1,1,0],[9E+09,9E+09,9E+09,9E+09,9E+09,9E+09]];
    CONST robtarget Target_1460:=[[231.497666319,-34.15081374,-16],[0,0.97236992,0,-0.233445365],[-2,-1,1,0],[9E+09,9E+09,9E+09,9E+09,9E+09,9E+09]];
    CONST robtarget Target_1470:=[[226.710430165,-37.900820893,-16],[0,0.97236992,0,-0.233445365],[-2,-1,1,0],[9E+09,9E+09,9E+09,9E+09,9E+09,9E+09]];
    CONST robtarget Target_1480:=[[226.710430165,-43.525820893,-16],[0,0.97236992,0,-0.233445365],[-2,-1,1,0],[9E+09,9E+09,9E+09,9E+09,9E+09,9E+09]];
    CONST robtarget Target_1490:=[[231.497666319,-42.58831374,-16],[0,0.97236992,0,-0.233445365],[-2,-1,1,0],[9E+09,9E+09,9E+09,9E+09,9E+09,9E+09]];
    CONST robtarget Target_1500:=[[237.242346485,-35.088320893,-16],[0,0.97236992,0,-0.233445365],[-2,-1,1,0],[9E+09,9E+09,9E+09,9E+09,9E+09,9E+09]];
    CONST robtarget Target_1510:=[[237.242346485,-17.27581374,-16],[0,0.97236992,0,-0.233445365],[-2,-1,1,0],[9E+09,9E+09,9E+09,9E+09,9E+09,9E+09]];
    CONST robtarget Target_1520:=[[231.497666319,-9.775820893,-16],[0,0.97236992,0,-0.233445365],[-2,-1,1,0],[9E+09,9E+09,9E+09,9E+09,9E+09,9E+09]];
    CONST robtarget Target_1530:=[[222.880643387,-6.963320893,-16],[0,0.97236992,0,-0.233445365],[-2,-1,1,0],[9E+09,9E+09,9E+09,9E+09,9E+09,9E+09]];
    CONST robtarget Target_1530_2:=[[222.880643387,-6.963320893,9],[0,0.97236992,0,-0.233445365],[-2,-1,1,0],[9E+09,9E+09,9E+09,9E+09,9E+09,9E+09]];
    CONST robtarget Target_1540:=[[193.199793179,-51.02581374,-16],[0,0.97236992,0,-0.233445365],[-2,-1,1,0],[9E+09,9E+09,9E+09,9E+09,9E+09,9E+09]];
    CONST robtarget Target_1550:=[[238.199793179,-51.02581374,-16],[0,0.97236992,0,-0.233445365],[-2,-1,1,0],[9E+09,9E+09,9E+09,9E+09,9E+09,9E+09]];
    CONST robtarget Target_1560:=[[238.199793179,-56.65081374,-16],[0,0.97236992,0,-0.233445365],[-2,-1,1,0],[9E+09,9E+09,9E+09,9E+09,9E+09,9E+09]];
    CONST robtarget Target_1570:=[[220.008303304,-56.65081374,-16],[0,0.97236992,0,-0.233445365],[-2,-1,1,0],[9E+09,9E+09,9E+09,9E+09,9E+09,9E+09]];
    CONST robtarget Target_1580:=[[220.008303304,-82.900820893,-16],[0,0.97236992,0,-0.233445365],[-2,-1,1,0],[9E+09,9E+09,9E+09,9E+09,9E+09,9E+09]];
    CONST robtarget Target_1590:=[[238.199793179,-82.900820893,-16],[0,0.97236992,0,-0.233445365],[-2,-1,1,0],[9E+09,9E+09,9E+09,9E+09,9E+09,9E+09]];
    CONST robtarget Target_1600:=[[238.199793179,-88.525810164,-16],[0,0.97236992,0,-0.233445365],[-2,-1,1,0],[9E+09,9E+09,9E+09,9E+09,9E+09,9E+09]];
    CONST robtarget Target_1610:=[[193.199793179,-88.525810164,-16],[0,0.97236992,0,-0.233445365],[-2,-1,1,0],[9E+09,9E+09,9E+09,9E+09,9E+09,9E+09]];
    CONST robtarget Target_1620:=[[193.199793179,-82.900820893,-16],[0,0.97236992,0,-0.233445365],[-2,-1,1,0],[9E+09,9E+09,9E+09,9E+09,9E+09,9E+09]];
    CONST robtarget Target_1630:=[[214.263623138,-82.900820893,-16],[0,0.97236992,0,-0.233445365],[-2,-1,1,0],[9E+09,9E+09,9E+09,9E+09,9E+09,9E+09]];
    CONST robtarget Target_1640:=[[214.263623138,-56.65081374,-16],[0,0.97236992,0,-0.233445365],[-2,-1,1,0],[9E+09,9E+09,9E+09,9E+09,9E+09,9E+09]];
    CONST robtarget Target_1650:=[[193.199793179,-56.65081374,-16],[0,0.97236992,0,-0.233445365],[-2,-1,1,0],[9E+09,9E+09,9E+09,9E+09,9E+09,9E+09]];
    CONST robtarget Target_1660:=[[193.199793179,-51.02581374,-16],[0,0.97236992,0,-0.233445365],[-2,-1,1,0],[9E+09,9E+09,9E+09,9E+09,9E+09,9E+09]];
    CONST robtarget Target_1660_2:=[[193.199793179,-51.02581374,9],[0,0.97236992,0,-0.233445365],[-2,-1,1,0],[9E+09,9E+09,9E+09,9E+09,9E+09,9E+09]];
    PROC main()
        MoveL Target_10_2,v100,fine,My_Mechanism_2\WObj:=Minor_1;
        MoveL Target_10,v100,fine,My_Mechanism_2\WObj:=Minor_1;
        MoveL Target_20,v100,fine,My_Mechanism_2\WObj:=Minor_1;
        MoveL Target_30,v100,fine,My_Mechanism_2\WObj:=Minor_1;
        MoveL Target_40,v100,fine,My_Mechanism_2\WObj:=Minor_1;
        MoveL Target_50,v100,fine,My_Mechanism_2\WObj:=Minor_1;
        MoveL Target_10_2,v100,fine,My_Mechanism_2\WObj:=Minor_1;
        MoveL Target_60,v100,fine,My_Mechanism_2\WObj:=Minor_1;
        MoveL Target_70,v100,fine,My_Mechanism_2\WObj:=Minor_1;
        MoveL Target_80,v100,fine,My_Mechanism_2\WObj:=Minor_1;
        MoveL Target_90,v100,fine,My_Mechanism_2\WObj:=Minor_1;
        MoveL Target_100,v100,fine,My_Mechanism_2\WObj:=Minor_1;
        MoveL Target_100_2,v100,fine,My_Mechanism_2\WObj:=Minor_1;
        MoveL Target_110,v100,fine,My_Mechanism_2\WObj:=Minor_1;
        MoveL Target_120,v100,fine,My_Mechanism_2\WObj:=Minor_1;
        MoveL Target_130,v100,fine,My_Mechanism_2\WObj:=Minor_1;
        MoveL Target_140,v100,fine,My_Mechanism_2\WObj:=Minor_1;
        MoveL Target_150,v100,fine,My_Mechanism_2\WObj:=Minor_1;
        MoveL Target_160,v100,fine,My_Mechanism_2\WObj:=Minor_1;
        MoveL Target_170,v100,fine,My_Mechanism_2\WObj:=Minor_1;
        MoveL Target_180,v100,fine,My_Mechanism_2\WObj:=Minor_1;
        MoveL Target_190,v100,fine,My_Mechanism_2\WObj:=Minor_1;
        MoveL Target_200,v100,fine,My_Mechanism_2\WObj:=Minor_1;
        MoveL Target_210,v100,fine,My_Mechanism_2\WObj:=Minor_1;
        MoveL Target_220,v100,fine,My_Mechanism_2\WObj:=Minor_1;
        MoveL Target_230,v100,fine,My_Mechanism_2\WObj:=Minor_1;
        MoveL Target_230_2,v100,fine,My_Mechanism_2\WObj:=Minor_1;
        MoveL Target_240,v100,fine,My_Mechanism_2\WObj:=Minor_1;
        MoveL Target_250,v100,fine,My_Mechanism_2\WObj:=Minor_1;
        MoveL Target_260,v100,fine,My_Mechanism_2\WObj:=Minor_1;
        MoveL Target_270,v100,fine,My_Mechanism_2\WObj:=Minor_1;
        MoveL Target_280,v100,fine,My_Mechanism_2\WObj:=Minor_1;
        MoveL Target_290,v100,fine,My_Mechanism_2\WObj:=Minor_1;
        MoveL Target_300,v100,fine,My_Mechanism_2\WObj:=Minor_1;
        MoveL Target_310,v100,fine,My_Mechanism_2\WObj:=Minor_1;
        MoveL Target_320,v100,fine,My_Mechanism_2\WObj:=Minor_1;
        MoveL Target_330,v100,fine,My_Mechanism_2\WObj:=Minor_1;
        MoveL Target_340,v100,fine,My_Mechanism_2\WObj:=Minor_1;
        MoveL Target_350,v100,fine,My_Mechanism_2\WObj:=Minor_1;
        MoveL Target_360,v100,fine,My_Mechanism_2\WObj:=Minor_1;
        MoveL Target_370,v100,fine,My_Mechanism_2\WObj:=Minor_1;
        MoveL Target_370_2,v100,fine,My_Mechanism_2\WObj:=Minor_1;
        MoveL Target_380,v100,fine,My_Mechanism_2\WObj:=Minor_1;
        MoveL Target_390,v100,fine,My_Mechanism_2\WObj:=Minor_1;
        MoveL Target_400,v100,fine,My_Mechanism_2\WObj:=Minor_1;
        MoveL Target_410,v100,fine,My_Mechanism_2\WObj:=Minor_1;
        MoveL Target_420,v100,fine,My_Mechanism_2\WObj:=Minor_1;
        MoveL Target_430,v100,fine,My_Mechanism_2\WObj:=Minor_1;
        MoveL Target_440,v100,fine,My_Mechanism_2\WObj:=Minor_1;
        MoveL Target_450,v100,fine,My_Mechanism_2\WObj:=Minor_1;
        MoveL Target_460,v100,fine,My_Mechanism_2\WObj:=Minor_1;
        MoveL Target_470,v100,fine,My_Mechanism_2\WObj:=Minor_1;
        MoveL Target_480,v100,fine,My_Mechanism_2\WObj:=Minor_1;
        MoveL Target_480_2,v100,fine,My_Mechanism_2\WObj:=Minor_1;
        MoveL Target_490,v100,fine,My_Mechanism_2\WObj:=Minor_1;
        MoveL Target_500,v100,fine,My_Mechanism_2\WObj:=Minor_1;
        MoveL Target_510,v100,fine,My_Mechanism_2\WObj:=Minor_1;
        MoveL Target_520,v100,fine,My_Mechanism_2\WObj:=Minor_1;
        MoveL Target_530,v100,fine,My_Mechanism_2\WObj:=Minor_1;
        MoveL Target_540,v100,fine,My_Mechanism_2\WObj:=Minor_1;
        MoveL Target_550,v100,fine,My_Mechanism_2\WObj:=Minor_1;
        MoveL Target_560,v100,fine,My_Mechanism_2\WObj:=Minor_1;
        MoveL Target_570,v100,fine,My_Mechanism_2\WObj:=Minor_1;
        MoveL Target_580,v100,fine,My_Mechanism_2\WObj:=Minor_1;
        MoveL Target_590,v100,fine,My_Mechanism_2\WObj:=Minor_1;
        MoveL Target_600,v100,fine,My_Mechanism_2\WObj:=Minor_1;
        MoveL Target_610,v100,fine,My_Mechanism_2\WObj:=Minor_1;
        MoveL Target_620,v100,fine,My_Mechanism_2\WObj:=Minor_1;
        MoveL Target_630,v100,fine,My_Mechanism_2\WObj:=Minor_1;
        MoveL Target_640,v100,fine,My_Mechanism_2\WObj:=Minor_1;
        MoveL Target_640_2,v100,fine,My_Mechanism_2\WObj:=Minor_1;
        MoveL Target_650,v100,fine,My_Mechanism_2\WObj:=Minor_1;
        MoveL Target_660,v100,fine,My_Mechanism_2\WObj:=Minor_1;
        MoveL Target_670,v100,fine,My_Mechanism_2\WObj:=Minor_1;
        MoveL Target_680,v100,fine,My_Mechanism_2\WObj:=Minor_1;
        MoveL Target_690,v100,fine,My_Mechanism_2\WObj:=Minor_1;
        MoveL Target_700,v100,fine,My_Mechanism_2\WObj:=Minor_1;
        MoveL Target_710,v100,fine,My_Mechanism_2\WObj:=Minor_1;
        MoveL Target_720,v100,fine,My_Mechanism_2\WObj:=Minor_1;
        MoveL Target_730,v100,fine,My_Mechanism_2\WObj:=Minor_1;
        MoveL Target_730_2,v100,fine,My_Mechanism_2\WObj:=Minor_1;
        MoveL Target_740,v100,fine,My_Mechanism_2\WObj:=Minor_1;
        MoveL Target_750,v100,fine,My_Mechanism_2\WObj:=Minor_1;
        MoveL Target_760,v100,fine,My_Mechanism_2\WObj:=Minor_1;
        MoveL Target_770,v100,fine,My_Mechanism_2\WObj:=Minor_1;
        MoveL Target_770_2,v100,fine,My_Mechanism_2\WObj:=Minor_1;
        MoveL Target_780,v100,fine,My_Mechanism_2\WObj:=Minor_1;
        MoveL Target_790,v100,fine,My_Mechanism_2\WObj:=Minor_1;
        MoveL Target_800,v100,fine,My_Mechanism_2\WObj:=Minor_1;
        MoveL Target_810,v100,fine,My_Mechanism_2\WObj:=Minor_1;
        MoveL Target_820,v100,fine,My_Mechanism_2\WObj:=Minor_1;
        MoveL Target_830,v100,fine,My_Mechanism_2\WObj:=Minor_1;
        MoveL Target_840,v100,fine,My_Mechanism_2\WObj:=Minor_1;
        MoveL Target_850,v100,fine,My_Mechanism_2\WObj:=Minor_1;
        MoveL Target_860,v100,fine,My_Mechanism_2\WObj:=Minor_1;
        MoveL Target_870,v100,fine,My_Mechanism_2\WObj:=Minor_1;
        MoveL Target_880,v100,fine,My_Mechanism_2\WObj:=Minor_1;
        MoveL Target_880_2,v100,fine,My_Mechanism_2\WObj:=Minor_1;
        MoveL Target_890,v100,fine,My_Mechanism_2\WObj:=Minor_1;
        MoveL Target_900,v100,fine,My_Mechanism_2\WObj:=Minor_1;
        MoveL Target_910,v100,fine,My_Mechanism_2\WObj:=Minor_1;
        MoveL Target_920,v100,fine,My_Mechanism_2\WObj:=Minor_1;
        MoveL Target_930,v100,fine,My_Mechanism_2\WObj:=Minor_1;
        MoveL Target_940,v100,fine,My_Mechanism_2\WObj:=Minor_1;
        MoveL Target_950,v100,fine,My_Mechanism_2\WObj:=Minor_1;
        MoveL Target_960,v100,fine,My_Mechanism_2\WObj:=Minor_1;
        MoveL Target_970,v100,fine,My_Mechanism_2\WObj:=Minor_1;
        MoveL Target_980,v100,fine,My_Mechanism_2\WObj:=Minor_1;
        MoveL Target_990,v100,fine,My_Mechanism_2\WObj:=Minor_1;
        MoveL Target_1000,v100,fine,My_Mechanism_2\WObj:=Minor_1;
        MoveL Target_1010,v100,fine,My_Mechanism_2\WObj:=Minor_1;
        MoveL Target_1020,v100,fine,My_Mechanism_2\WObj:=Minor_1;
        MoveL Target_1030,v100,fine,My_Mechanism_2\WObj:=Minor_1;
        MoveL Target_1040,v100,fine,My_Mechanism_2\WObj:=Minor_1;
        MoveL Target_1050,v100,fine,My_Mechanism_2\WObj:=Minor_1;
        MoveL Target_1060,v100,fine,My_Mechanism_2\WObj:=Minor_1;
        MoveL Target_1070,v100,fine,My_Mechanism_2\WObj:=Minor_1;
        MoveL Target_1080,v100,fine,My_Mechanism_2\WObj:=Minor_1;
        MoveL Target_1090,v100,fine,My_Mechanism_2\WObj:=Minor_1;
        MoveL Target_1100,v100,fine,My_Mechanism_2\WObj:=Minor_1;
        MoveL Target_1110,v100,fine,My_Mechanism_2\WObj:=Minor_1;
        MoveL Target_1120,v100,fine,My_Mechanism_2\WObj:=Minor_1;
        MoveL Target_1130,v100,fine,My_Mechanism_2\WObj:=Minor_1;
        MoveL Target_1130_2,v100,fine,My_Mechanism_2\WObj:=Minor_1;
        MoveL Target_1140,v100,fine,My_Mechanism_2\WObj:=Minor_1;
        MoveL Target_1150,v100,fine,My_Mechanism_2\WObj:=Minor_1;
        MoveL Target_1160,v100,fine,My_Mechanism_2\WObj:=Minor_1;
        MoveL Target_1170,v100,fine,My_Mechanism_2\WObj:=Minor_1;
        MoveL Target_1180,v100,fine,My_Mechanism_2\WObj:=Minor_1;
        MoveL Target_1180_2,v100,fine,My_Mechanism_2\WObj:=Minor_1;
        MoveL Target_1190,v100,fine,My_Mechanism_2\WObj:=Minor_1;
        MoveL Target_1200,v100,fine,My_Mechanism_2\WObj:=Minor_1;
        MoveL Target_1210,v100,fine,My_Mechanism_2\WObj:=Minor_1;
        MoveL Target_1220,v100,fine,My_Mechanism_2\WObj:=Minor_1;
        MoveL Target_1230,v100,fine,My_Mechanism_2\WObj:=Minor_1;
        MoveL Target_1240,v100,fine,My_Mechanism_2\WObj:=Minor_1;
        MoveL Target_1250,v100,fine,My_Mechanism_2\WObj:=Minor_1;
        MoveL Target_1260,v100,fine,My_Mechanism_2\WObj:=Minor_1;
        MoveL Target_1270,v100,fine,My_Mechanism_2\WObj:=Minor_1;
        MoveL Target_1280,v100,fine,My_Mechanism_2\WObj:=Minor_1;
        MoveL Target_1290,v100,fine,My_Mechanism_2\WObj:=Minor_1;
        MoveL Target_1290_2,v100,fine,My_Mechanism_2\WObj:=Minor_1;
        MoveL Target_1300,v100,fine,My_Mechanism_2\WObj:=Minor_1;
        MoveL Target_1310,v100,fine,My_Mechanism_2\WObj:=Minor_1;
        MoveL Target_1320,v100,fine,My_Mechanism_2\WObj:=Minor_1;
        MoveL Target_1330,v100,fine,My_Mechanism_2\WObj:=Minor_1;
        MoveL Target_1340,v100,fine,My_Mechanism_2\WObj:=Minor_1;
        MoveL Target_1350,v100,fine,My_Mechanism_2\WObj:=Minor_1;
        MoveL Target_1360,v100,fine,My_Mechanism_2\WObj:=Minor_1;
        MoveL Target_1370,v100,fine,My_Mechanism_2\WObj:=Minor_1;
        MoveL Target_1380,v100,fine,My_Mechanism_2\WObj:=Minor_1;
        MoveL Target_1390,v100,fine,My_Mechanism_2\WObj:=Minor_1;
        MoveL Target_1400,v100,fine,My_Mechanism_2\WObj:=Minor_1;
        MoveL Target_1410,v100,fine,My_Mechanism_2\WObj:=Minor_1;
        MoveL Target_1420,v100,fine,My_Mechanism_2\WObj:=Minor_1;
        MoveL Target_1430,v100,fine,My_Mechanism_2\WObj:=Minor_1;
        MoveL Target_1440,v100,fine,My_Mechanism_2\WObj:=Minor_1;
        MoveL Target_1450,v100,fine,My_Mechanism_2\WObj:=Minor_1;
        MoveL Target_1460,v100,fine,My_Mechanism_2\WObj:=Minor_1;
        MoveL Target_1470,v100,fine,My_Mechanism_2\WObj:=Minor_1;
        MoveL Target_1480,v100,fine,My_Mechanism_2\WObj:=Minor_1;
        MoveL Target_1490,v100,fine,My_Mechanism_2\WObj:=Minor_1;
        MoveL Target_1500,v100,fine,My_Mechanism_2\WObj:=Minor_1;
        MoveL Target_1510,v100,fine,My_Mechanism_2\WObj:=Minor_1;
        MoveL Target_1520,v100,fine,My_Mechanism_2\WObj:=Minor_1;
        MoveL Target_1530,v100,fine,My_Mechanism_2\WObj:=Minor_1;
        MoveL Target_1530_2,v100,fine,My_Mechanism_2\WObj:=Minor_1;
        MoveL Target_1540,v100,fine,My_Mechanism_2\WObj:=Minor_1;
        MoveL Target_1550,v100,fine,My_Mechanism_2\WObj:=Minor_1;
        MoveL Target_1560,v100,fine,My_Mechanism_2\WObj:=Minor_1;
        MoveL Target_1570,v100,fine,My_Mechanism_2\WObj:=Minor_1;
        MoveL Target_1580,v100,fine,My_Mechanism_2\WObj:=Minor_1;
        MoveL Target_1590,v100,fine,My_Mechanism_2\WObj:=Minor_1;
        MoveL Target_1600,v100,fine,My_Mechanism_2\WObj:=Minor_1;
        MoveL Target_1610,v100,fine,My_Mechanism_2\WObj:=Minor_1;
        MoveL Target_1620,v100,fine,My_Mechanism_2\WObj:=Minor_1;
        MoveL Target_1630,v100,fine,My_Mechanism_2\WObj:=Minor_1;
        MoveL Target_1640,v100,fine,My_Mechanism_2\WObj:=Minor_1;
        MoveL Target_1650,v100,fine,My_Mechanism_2\WObj:=Minor_1;
        MoveL Target_1660,v100,fine,My_Mechanism_2\WObj:=Minor_1;
        MoveL Target_1660_2,v100,fine,My_Mechanism_2\WObj:=Minor_1;
    ENDPROC
ENDMODULE

--- Backups/Controller8/RAPID/TASK1/SYSMOD/LINKEDM.sys ---
%%%
  VERSION:1
  LANGUAGE:ENGLISH
%%%

MODULE LINKEDM (SYSMODULE)

! FOLLOWER
!     Name of electronically linked follower axis used by operator at teach pendent.
      PERS string l_f_axis_name{5}       :=  ["",  "", "", "", ""];

!     Name of the mechanical unit for follower axis.
      PERS string l_f_mecunt_n{5}  :=  ["", "", "", "", ""];

!     Linked follower axis number in the mechanical unit (first axis in mech. unit is number 1).
      PERS num l_f_axis_no{5}      :=  [0,          0,   0,  0,  0];

! MASTER
!     Name of the mechanical unit for linked master axis.
      PERS string l_m_mecunt_n{5} :=  ["", "", "", "", ""];

!     Linked master axis number in the mechanical unit (first axis in mech. unit is number 1).
!     See axis number table in documentation for different master mechanical units.
      PERS num l_m_axis_no{5}     :=  [0,  0,  0,  0,  0];

! POSITION OFFSET
!     The increase of the allowed offset position between the master and follower
!     positions, used when starting AUTO mode. As soon as the offset is decreased
!     the old configurated parameter is used.
!     Example: 3 => the configurated value of allowed offset is increased 3 times.
      PERS num offset_ratio{5}       :=  [10,  10,   10,  10,  10];

! SPEED RATIO
!     Speed_ratio used in AUTO and JOG modes [ very_slow   slow    normal    fast]
!     Value 1 = max allowed manual speed.
      CONST num speed_ratio {20}      := [0.01, 0.01, 0.01, 0.01, 0.01,
                                          0.05, 0.05, 0.05, 0.05, 0.05,
                                          0.20, 0.20, 0.20, 0.20, 0.20,
                                          1.00, 1.00, 1.00, 1.00, 1.00];

! STEP SIZE
!     Displacement position used in JOG mode for each activation of positive or
!     negative movement.                  [very_short    short   normal   long]
!     Unit degees or meter.
      CONST num displacement {20}     := [0.001, 0.001, 0.001, 0.001, 0.001,
                                          0.005, 0.005, 0.005, 0.005, 0.005,
                                          0.020, 0.020, 0.020, 0.020, 0.020,
                                          0.100, 0.100, 0.100, 0.100, 0.100];


!-------------------------------------------------------------
 PROC Linked_m ()
      Linked_m_exe ;
 ENDPROC
ENDMODULE
